PROGRAM P_ADS_OEE
VAR
	btonDelayAfterStart :BOOL;
	fbRead_1: FB_ReadAdsSymByName;	
	fbCyclicReadout: TON;
	uiCounterGoodBottles :UINT;
	fbRead_2: FB_ReadAdsSymByName;
	AStBadPackageReason  :ARRAY[0..63] OF S_Information;
	fbRead_3: FB_ReadAdsSymByName;
	uiCounterBadBottles  :UINT;
	fbRead_4: FB_ReadAdsSymByName;
	fbRead_5: FB_ReadAdsSymByName;
	bCycleReset :BOOL;
	udiCounterExecuteTime :UINT;
	fbRead_6: FB_ReadAdsSymByName;
	btonConfectionEnding:BOOL;
	fbRead_7: FB_ReadAdsSymByName;
	
END_VAR

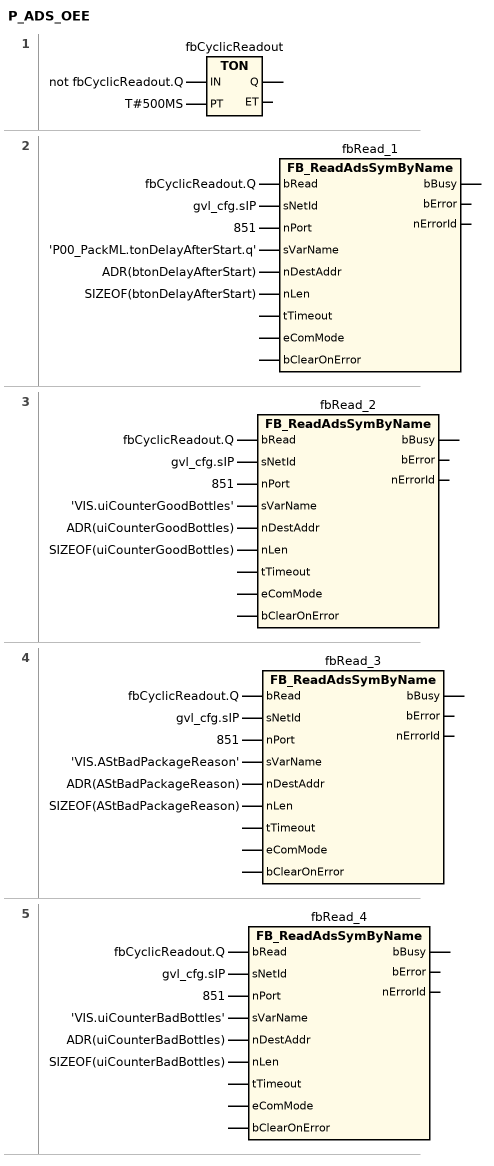
// NETWORK 1
fbCyclicReadout(IN := not fbCyclicReadout.Q, PT := T#500MS); // TON

// NETWORK 2
fbRead_1(
    bRead := fbCyclicReadout.Q,
    sNetId := gvl_cfg.sIP,
    nPort := 851,
    sVarName := 'P00_PackML.tonDelayAfterStart.q',
    nDestAddr := ADR(btonDelayAfterStart),
    nLen := SIZEOF(btonDelayAfterStart)); // FB_ReadAdsSymByName

// NETWORK 3
fbRead_2(
    bRead := fbCyclicReadout.Q,
    sNetId := gvl_cfg.sIP,
    nPort := 851,
    sVarName := 'VIS.uiCounterGoodBottles',
    nDestAddr := ADR(uiCounterGoodBottles),
    nLen := SIZEOF(uiCounterGoodBottles)); // FB_ReadAdsSymByName

// NETWORK 4
fbRead_3(
    bRead := fbCyclicReadout.Q,
    sNetId := gvl_cfg.sIP,
    nPort := 851,
    sVarName := 'VIS.AStBadPackageReason',
    nDestAddr := ADR(AStBadPackageReason),
    nLen := SIZEOF(AStBadPackageReason)); // FB_ReadAdsSymByName

// NETWORK 5
fbRead_4(
    bRead := fbCyclicReadout.Q,
    sNetId := gvl_cfg.sIP,
    nPort := 851,
    sVarName := 'VIS.uiCounterBadBottles',
    nDestAddr := ADR(uiCounterBadBottles),
    nLen := SIZEOF(uiCounterBadBottles)); // FB_ReadAdsSymByName

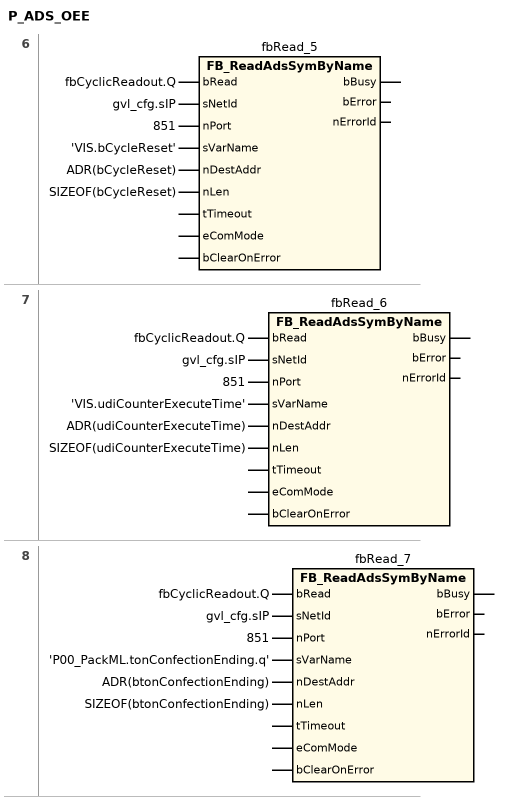
// NETWORK 6
fbRead_5(
    bRead := fbCyclicReadout.Q,
    sNetId := gvl_cfg.sIP,
    nPort := 851,
    sVarName := 'VIS.bCycleReset',
    nDestAddr := ADR(bCycleReset),
    nLen := SIZEOF(bCycleReset)); // FB_ReadAdsSymByName

// NETWORK 7
fbRead_6(
    bRead := fbCyclicReadout.Q,
    sNetId := gvl_cfg.sIP,
    nPort := 851,
    sVarName := 'VIS.udiCounterExecuteTime',
    nDestAddr := ADR(udiCounterExecuteTime),
    nLen := SIZEOF(udiCounterExecuteTime)); // FB_ReadAdsSymByName

// NETWORK 8
fbRead_7(
    bRead := fbCyclicReadout.Q,
    sNetId := gvl_cfg.sIP,
    nPort := 851,
    sVarName := 'P00_PackML.tonConfectionEnding.q',
    nDestAddr := ADR(btonConfectionEnding),
    nLen := SIZEOF(btonConfectionEnding)); // FB_ReadAdsSymByName

END_PROGRAM

(* stored: Version 1.1.0.1, ProductVersion 3.1.4026.13, FileIdentifier eca1fbe5534909898b0a3cdb4f90d8bc0634fac8, FileSignature a4642d525bba0b025314b36a799c82395388e3ab11c474fd22b965f6c5d430ac64a942d617cd972563f28555bee463352bb67cb92614604880a2c6cd3886bd3b6c01360484a69038d76108636f0282d95f4fbd00cc2360d0c8e54e20ec86d2f32b9368a1276af5b57618f6662441e1d68930c54d4faecd8ac08623b2ed74f3152022ba30cd4f7771b6692f781a490f55219b832c343d88058766936b1675b0f58e0d34a8327855f5442b0344c03284ba365ea6177da1ee21b9bd0ef81b5c3e91b7eff3000179616b5a901170ddda7d72b5401022d57d2ade194de605c7df333b03185ee9812c5a5883e65fe920542aa5203049307d239b385b868287ea08eeae
   POU P_ADS_OEE: Id {3df42384-c158-490c-afe6-3585092a157d}, SpecialFunc None *)
